Staubli VAL3: EnterPageKey.pgx

program EnterPageKey(num& x_nKey, num& x_nSelect, string& x_sItem)
  local bool l_bRes
  local num l_nItem
  local num l_nKey
  local num l_nView
  local string l_sEmpty
  local string l_sItem
  local string l_sStr
  local string l_sTool
  local string l_sValue
  local string l_sYN[2]
  local point lp
begin
  //
  switch x_nSelect
    case 0
      if x_nKey==271
        uPallet[sItem].pO=here(tTool,world)
        popUpMsg("OK")
      endIf

    break
    case 1
      if x_nKey==271
        uPallet[sItem].pO=here(tTool,world)
        popUpMsg("OK")
      endIf

    break
    case 2
      if x_nKey==271
        uPallet[sItem].pO=here(tTool,world)
        popUpMsg("OK")
      endIf

    break

    case 3
      if x_nKey==270
        call user:editNum(x_sItem,sListItemValue[x_nSelect],uPallet[sItem].ndX,x_nSelect)
      endIf
    break
    case 4
      if x_nKey==270
        call user:editNum(x_sItem,sListItemValue[x_nSelect],uPallet[sItem].ndY,x_nSelect)
      endIf
    break

    case 5
      if x_nKey==271
        if setFrame(pPonit[0],pPonit[1],pPonit[2],fFrame)==0
          uPallet[sItem].pStart=here(tTool,fFrame)
          popUpMsg("OK")
        else
          uPallet[sItem].pStart=here(tTool,fFrame)
          popUpMsg("请先记录原点，X点和Y点！")
        endIf
      endIf
    break

  endSwitch
  //
  if x_nKey==272
    call Tool:Main(1)
    call Tool:getTool(l_sTool,tTool)
    if l_sTool!=""
      uPallet[sItem].sToolName=l_sTool
      sParameter[6]="工具"
      sListItemValue[6]=uPallet[sItem].sToolName
      call user:strlength(sParameter[6],user:nBottomX/2)
      l_sValue=sListItemValue[6]
      call user:strlength(l_sValue,user:nBottomX/2+1)
      sParameter[6]=sParameter[6]+":"+l_sValue
    endIf
    if x_nKey==270 or x_nKey==272
      bUserRefresh=true
      bListRefresh=true
    endIf
  endIf

end
